# EPICS autosave request: ADPerkinElmer/iocs/perkinElmerIOC/iocBoot/iocPerkinElmer/auto_settings.req
file "PerkinElmer_settings.req",  P=$(P),  R=cam1:
file "ADBase_settings.req",       P=$(P),  R=cam1:
file "NDPluginBase_settings.req", P=$(P),  R=image1:
file "NDStdArrays_settings.req",  P=$(P),  R=image1:
file "commonPlugin_settings.req", P=$(P)
